{attribute 'qualified_only' := ''}
VAR_GLOBAL
	///Realsubject class instance
	globalSubjectInstance: Realsubject;
END_VAR

(* stored: Version 1.1.0.1, ProductVersion 3.1.4024.12
   GVL GVL: Id {70a67f79-b967-4931-9d3f-ea67b822d4cf} *)
